PROGRAM PRG_CommWaage
	VAR
		ControllerWaage : SerialLineControl;
		nCount : DINT := 0;
END_VAR

ControllerWaage(
	Mode:= SERIALLINEMODE_EL6_22B, 
	pComIn:= ADR(ELDataIn_Waage), 
	pComOut:= ADR(ELDataOut_Waage), 
	SizeComIn:= TO_UINT( SIZEOF(ELDataIn_Waage)), 
	Error=> ErrorFastWaage, 
	ErrorID=> , 
	TxBuffer:= TxBufferWaage, 
	RxBuffer:= RxBufferWaage);
	
	nCount := nCount + 1;

END_PROGRAM

(* stored: Version 1.1.0.1, ProductVersion 3.1.4024.6
   POU PRG_CommWaage: Id {7cd68caf-d9da-4019-afd2-c32c2d58570e}, SpecialFunc None *)
